TYPE InputBase_8311D824 :
STRUCT
END_STRUCT
END_TYPE

(* stored: Version 1.2.0.0, ProductVersion 3.1.4024.12
   DUT InputBase_8311D824: Id {fc47fb74-3ed0-0064-25f7-7b1923007783} *)
